FUNCTION_BLOCK FbStateCoilFaultCoil
VAR_INPUT
	xTrigger: BOOL;
	xBreakCondition: BOOL;
END_VAR
VAR_OUTPUT
	xMemoryCoil: BOOL;
END_VAR

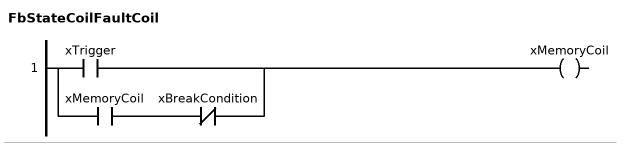
// NETWORK 1
xMemoryCoil := xTrigger OR xMemoryCoil AND NOT xBreakCondition;

END_FUNCTION_BLOCK

(* stored: Version 1.1.0.1, ProductVersion 3.1.4024.12
   POU FbStateCoilFaultCoil: Id {4d45d4a4-4eb9-47c4-9f69-bc63fb1800a3}, SpecialFunc None *)
